PROGRAM Axes
VAR
	Fb_MachX_Power: MC_Power;
	Fb_MachY_Power: MC_Power;
	Fb_MachZ_Power: MC_Power;
	Fb_SimsX_Power: MC_Power;
	Fb_SimsY_Power: MC_Power;
	Fb_SimsZ_Power: MC_Power;

	Fb_Axes_MachX_Reset: MC_Reset;
	Fb_Axes_MachY_Reset: MC_Reset;
	Fb_Axes_MachZ_Reset: MC_Reset;
	Fb_Axes_SimsX_Reset: MC_Reset;
	Fb_Axes_SimsY_Reset: MC_Reset;
	Fb_Axes_SimsZ_Reset: MC_Reset;
	
	fb_Axes_MachX_Jog: MC_Jog;
	fb_Axes_MachY_Jog: MC_Jog;
	fb_Axes_MachZ_Jog: MC_Jog;
	fb_Axes_SimsX_Jog: MC_Jog;
	fb_Axes_SimsY_Jog: MC_Jog;
	fb_Axes_SimsZ_Jog: MC_Jog;
	bo_override: BOOL;
	bo_tp_override: TP;
END_VAR

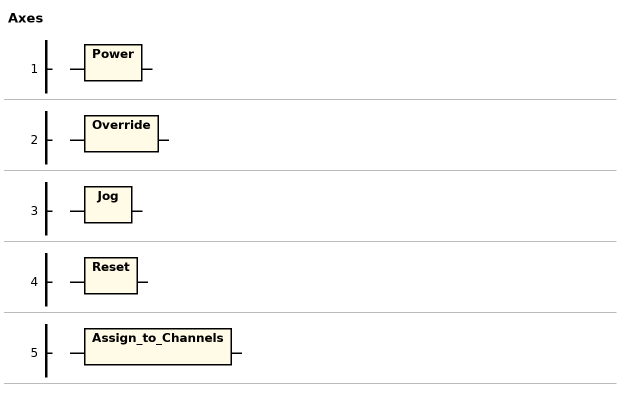
// NETWORK 1
Power();

// NETWORK 2
Override();

// NETWORK 3
Jog();

// NETWORK 4
Reset();

// NETWORK 5
Assign_to_Channels();

ACTION Assign_to_Channels:
st_Axes_Kin.nAxisIdsAcs[1]	:= MachX.NcToPlc.AxisId;
st_Axes_Kin.nAxisIdsAcs[2]	:= MachY.NcToPlc.AxisId;
st_Axes_Kin.nAxisIdsAcs[3]	:= MachZ.NcToPlc.AxisId;
st_Axes_Kin.nAxisIdsMcs[1]	:= SimsX.NcToPlc.AxisId;
st_Axes_Kin.nAxisIdsMcs[2]	:= SimsY.NcToPlc.AxisId;
st_Axes_Kin.nAxisIdsMcs[3]	:= SimsZ.NcToPlc.AxisId;
END_ACTION

ACTION Jog:
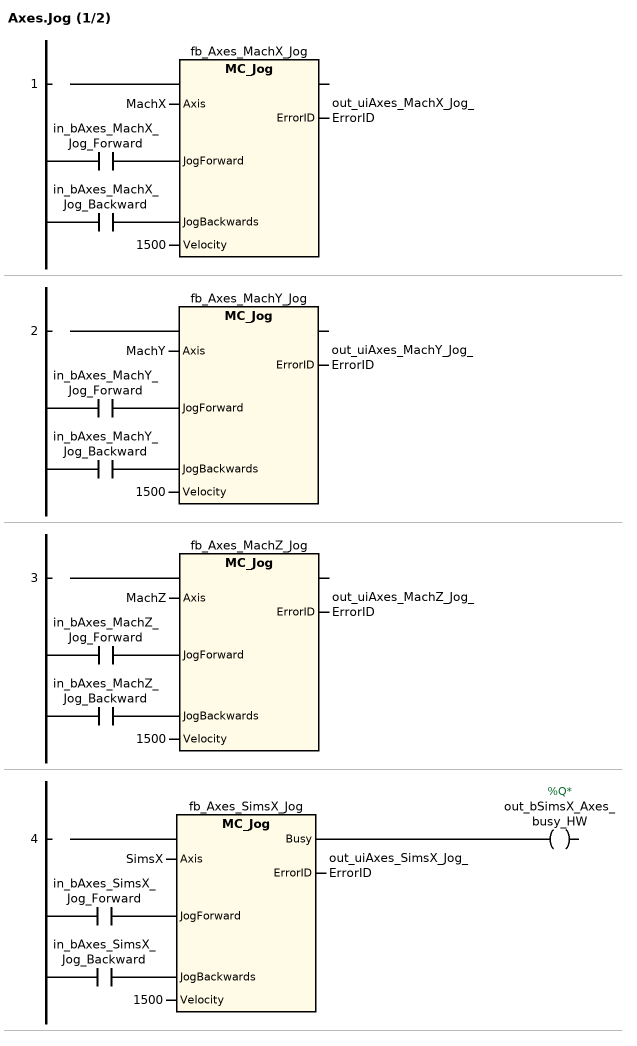
// NETWORK 1
fb_Axes_MachX_Jog(
    Axis := MachX,
    JogForward := in_bAxes_MachX_Jog_Forward,
    JogBackwards := in_bAxes_MachX_Jog_Backward,
    Velocity := 1500,
    ErrorID => out_uiAxes_MachX_Jog_ErrorID); // MC_Jog

// NETWORK 2
fb_Axes_MachY_Jog(
    Axis := MachY,
    JogForward := in_bAxes_MachY_Jog_Forward,
    JogBackwards := in_bAxes_MachY_Jog_Backward,
    Velocity := 1500,
    ErrorID => out_uiAxes_MachY_Jog_ErrorID); // MC_Jog

// NETWORK 3
fb_Axes_MachZ_Jog(
    Axis := MachZ,
    JogForward := in_bAxes_MachZ_Jog_Forward,
    JogBackwards := in_bAxes_MachZ_Jog_Backward,
    Velocity := 1500,
    ErrorID => out_uiAxes_MachZ_Jog_ErrorID); // MC_Jog

// NETWORK 4
//   out_bSimsX_Axes_busy_HW: AT %Q*
fb_Axes_SimsX_Jog(
    Axis := SimsX,
    JogForward := in_bAxes_SimsX_Jog_Forward,
    JogBackwards := in_bAxes_SimsX_Jog_Backward,
    Velocity := 1500,
    ErrorID => out_uiAxes_SimsX_Jog_ErrorID); // MC_Jog
out_bSimsX_Axes_busy_HW := fb_Axes_SimsX_Jog.Busy;

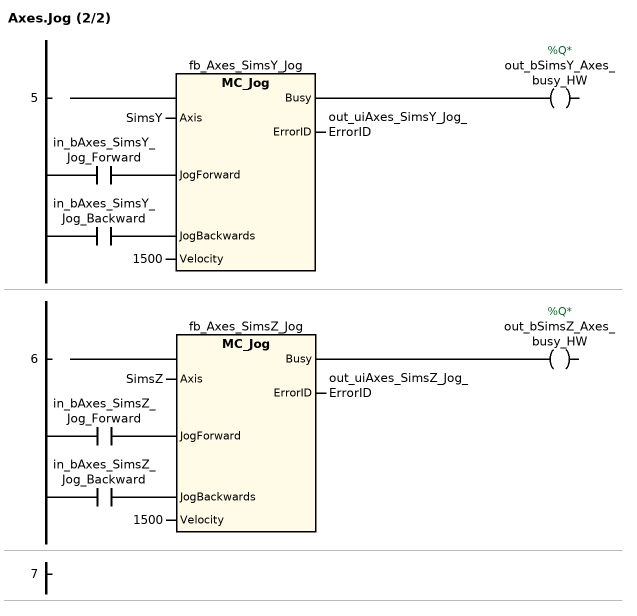
// NETWORK 5
//   out_bSimsY_Axes_busy_HW: AT %Q*
fb_Axes_SimsY_Jog(
    Axis := SimsY,
    JogForward := in_bAxes_SimsY_Jog_Forward,
    JogBackwards := in_bAxes_SimsY_Jog_Backward,
    Velocity := 1500,
    ErrorID => out_uiAxes_SimsY_Jog_ErrorID); // MC_Jog
out_bSimsY_Axes_busy_HW := fb_Axes_SimsY_Jog.Busy;

// NETWORK 6
//   out_bSimsZ_Axes_busy_HW: AT %Q*
fb_Axes_SimsZ_Jog(
    Axis := SimsZ,
    JogForward := in_bAxes_SimsZ_Jog_Forward,
    JogBackwards := in_bAxes_SimsZ_Jog_Backward,
    Velocity := 1500,
    ErrorID => out_uiAxes_SimsZ_Jog_ErrorID); // MC_Jog
out_bSimsZ_Axes_busy_HW := fb_Axes_SimsZ_Jog.Busy;

// NETWORK 7
END_ACTION

ACTION Override:
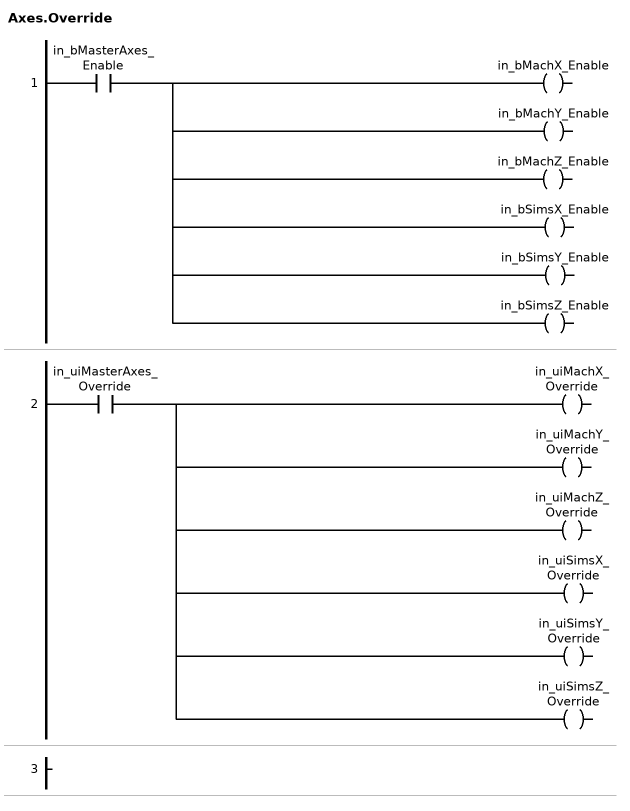
// NETWORK 1
in_bMachX_Enable := in_bMasterAxes_Enable;
in_bMachY_Enable := in_bMasterAxes_Enable;
in_bMachZ_Enable := in_bMasterAxes_Enable;
in_bSimsX_Enable := in_bMasterAxes_Enable;
in_bSimsY_Enable := in_bMasterAxes_Enable;
in_bSimsZ_Enable := in_bMasterAxes_Enable;

// NETWORK 2
in_uiMachX_Override := in_uiMasterAxes_Override;
in_uiMachY_Override := in_uiMasterAxes_Override;
in_uiMachZ_Override := in_uiMasterAxes_Override;
in_uiSimsX_Override := in_uiMasterAxes_Override;
in_uiSimsY_Override := in_uiMasterAxes_Override;
in_uiSimsZ_Override := in_uiMasterAxes_Override;

// NETWORK 3
END_ACTION

ACTION Power:
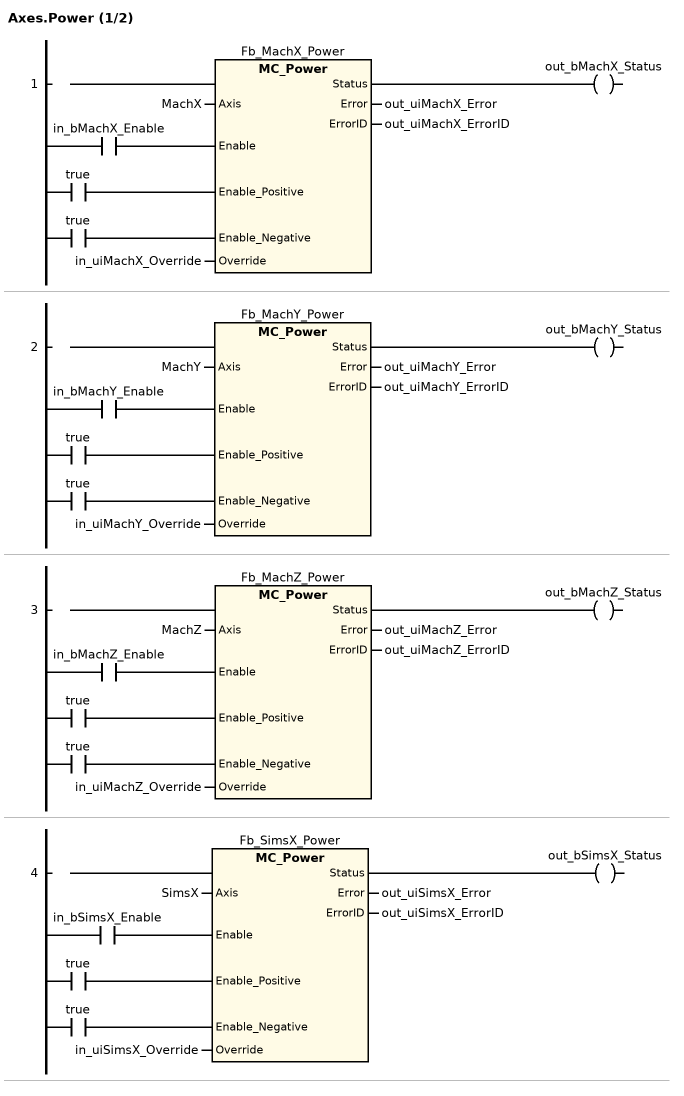
// NETWORK 1
Fb_MachX_Power(
    Axis := MachX,
    Enable := in_bMachX_Enable,
    Enable_Positive := true,
    Enable_Negative := true,
    Override := in_uiMachX_Override,
    Error => out_uiMachX_Error,
    ErrorID => out_uiMachX_ErrorID); // MC_Power
out_bMachX_Status := Fb_MachX_Power.Status;

// NETWORK 2
Fb_MachY_Power(
    Axis := MachY,
    Enable := in_bMachY_Enable,
    Enable_Positive := true,
    Enable_Negative := true,
    Override := in_uiMachY_Override,
    Error => out_uiMachY_Error,
    ErrorID => out_uiMachY_ErrorID); // MC_Power
out_bMachY_Status := Fb_MachY_Power.Status;

// NETWORK 3
Fb_MachZ_Power(
    Axis := MachZ,
    Enable := in_bMachZ_Enable,
    Enable_Positive := true,
    Enable_Negative := true,
    Override := in_uiMachZ_Override,
    Error => out_uiMachZ_Error,
    ErrorID => out_uiMachZ_ErrorID); // MC_Power
out_bMachZ_Status := Fb_MachZ_Power.Status;

// NETWORK 4
Fb_SimsX_Power(
    Axis := SimsX,
    Enable := in_bSimsX_Enable,
    Enable_Positive := true,
    Enable_Negative := true,
    Override := in_uiSimsX_Override,
    Error => out_uiSimsX_Error,
    ErrorID => out_uiSimsX_ErrorID); // MC_Power
out_bSimsX_Status := Fb_SimsX_Power.Status;

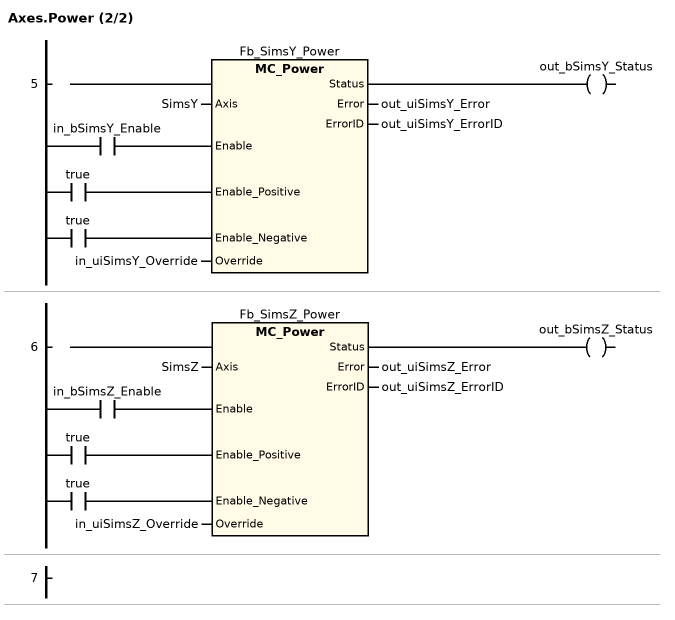
// NETWORK 5
Fb_SimsY_Power(
    Axis := SimsY,
    Enable := in_bSimsY_Enable,
    Enable_Positive := true,
    Enable_Negative := true,
    Override := in_uiSimsY_Override,
    Error => out_uiSimsY_Error,
    ErrorID => out_uiSimsY_ErrorID); // MC_Power
out_bSimsY_Status := Fb_SimsY_Power.Status;

// NETWORK 6
Fb_SimsZ_Power(
    Axis := SimsZ,
    Enable := in_bSimsZ_Enable,
    Enable_Positive := true,
    Enable_Negative := true,
    Override := in_uiSimsZ_Override,
    Error => out_uiSimsZ_Error,
    ErrorID => out_uiSimsZ_ErrorID); // MC_Power
out_bSimsZ_Status := Fb_SimsZ_Power.Status;

// NETWORK 7
END_ACTION

ACTION Reset:
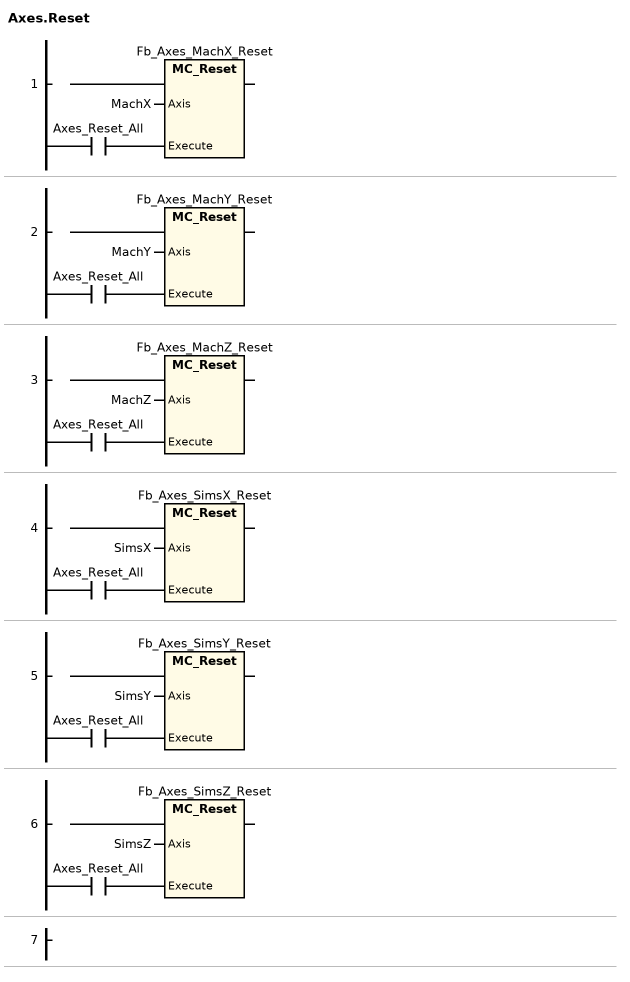
// NETWORK 1
Fb_Axes_MachX_Reset(Axis := MachX, Execute := Axes_Reset_All); // MC_Reset

// NETWORK 2
Fb_Axes_MachY_Reset(Axis := MachY, Execute := Axes_Reset_All); // MC_Reset

// NETWORK 3
Fb_Axes_MachZ_Reset(Axis := MachZ, Execute := Axes_Reset_All); // MC_Reset

// NETWORK 4
Fb_Axes_SimsX_Reset(Axis := SimsX, Execute := Axes_Reset_All); // MC_Reset

// NETWORK 5
Fb_Axes_SimsY_Reset(Axis := SimsY, Execute := Axes_Reset_All); // MC_Reset

// NETWORK 6
Fb_Axes_SimsZ_Reset(Axis := SimsZ, Execute := Axes_Reset_All); // MC_Reset

// NETWORK 7
END_ACTION

END_PROGRAM

(* stored: Version 1.1.0.1, ProductVersion 3.1.4018.9
   POU Axes: Id {0a42a9cb-90ba-466f-b3a4-4c16e7cbdc91}, SpecialFunc None
   Action Assign_to_Channels: Id {efc9eba8-6e65-4d90-8b48-2ad4d8dfc3e6}
   Action Jog: Id {a9e6cda4-ae91-4c44-a82e-2f38eedfcabb}
   Action Override: Id {4be583a9-8db5-4dd9-a9c9-a08e943c0186}
   Action Power: Id {0f98ef04-7193-44cb-86e0-afb4af112788}
   Action Reset: Id {deda37f8-2693-4b43-ad29-bee9734f07db} *)
